{attribute addProperty BoxType "EM7004-0000-9996"}
{attribute addProperty Id "Enable_PLSAT %Q*BOOL81"}
{attribute addProperty CRC "4128828442"}
{attribute addProperty SizeInBites "8"}
{attribute addProperty SizeInBytes "1"}
TYPE PLS_Outputs_F618EC1A :
STRUCT
	{attribute addProperty Name "Enable_PLS"}
	Enable_PLS AT %Q* : BOOL;
END_STRUCT
END_TYPE

(* stored: Version 1.2.0.0, ProductVersion 3.1.4024.9
   DUT PLS_Outputs_F618EC1A: Id {0b4654e9-d639-4e1f-beea-bae189ddcab3} *)
